FUNCTION_BLOCK Psd EXTENDS PlcModule
VAR_INPUT	
	Safety : Safety;
	
	{attribute 'OPC.UA.DA' := '0'}
	PsdConfig : PsdConfig;
	
	(* Axes *)
	IoStageAxis : IoStageAxis(Config := PsdConfig.AxesConfigs.IoStageAxisConfig);
	
	(* Chamber *)
	Chamber : PsdChamber(Config := PsdConfig.ChamberConfigs.PsdChamberConfig);
	
	(* Chuck *)
	Chuck : PsdChuck(Config := PsdConfig.ChuckConfigs.PsdChuckConfig);
	
	(* Ffu *)
	Ffu : Astrofan612Ffu(Config := PsdConfig.FfuConfigs.Astrofan612FfuConfig);
	
	(* Screen *)
	DM430GNScreenFS : DM430GNScreenFS(Config := PsdConfig.ScreenConfigs.DM430GNScreenConfigFS);
	DM430GNScreenBS : DM430GNScreenBS(Config := PsdConfig.ScreenConfigs.DM430GNScreenConfigBS);
	
	(* RFid *)
	Rfid : BisL405Rfid(Config := PsdConfig.RfidConfigs.BisL405RfidConfig);		
	
END_VAR
VAR_OUTPUT
END_VAR
VAR
END_VAR

SUPER^();

IF PsdConfig.SafetyIsEnabled THEN
	Safety();
END_IF

IF PsdConfig.AxesConfigs.IoStageAxisConfig.IsEnabled THEN
	IoStageAxis();	
END_IF

IF PsdConfig.ChamberConfigs.PsdChamberConfig.IsEnabled THEN
	Chamber();		
END_IF

IF PsdConfig.ChuckConfigs.PsdChuckConfig.IsEnabled THEN
	Chuck();		
END_IF

IF PsdConfig.FfuConfigs.Astrofan612FfuConfig.IsEnabled THEN
	Ffu();	
END_IF
	
// Screens
IF PsdConfig.ScreenConfigs.DM430GNScreenConfigFS.IsEnabled THEN
	DM430GNScreenFS();
	IF DM430GNScreenFS.InitConfigSerialCom THEN
		;
	END_IF
END_IF

IF PsdConfig.ScreenConfigs.DM430GNScreenConfigBS.IsEnabled THEN
	DM430GNScreenBS();
	IF DM430GNScreenBS.InitConfigSerialCom THEN
		;
	END_IF
END_IF

IF PsdConfig.RfidConfigs.BisL405RfidConfig.IsEnabled THEN
	Rfid();	
END_IF


IF IoStageAxis.GetPosition() = EStagePosition.Loading THEN
	Chamber.StageIsInLoadingPosition := TRUE;	
ELSE
	Chamber.StageIsInLoadingPosition := FALSE;
END_IF

METHOD FB_init : BOOL
VAR_INPUT
	bInitRetains : BOOL; // if TRUE, the retain variables are initialized (warm start / cold start)
	bInCopyCode : BOOL;  // if TRUE, the instance afterwards gets moved into the copy code (online change)
	Config : PsdConfig;
END_VAR
PsdConfig := Config;
PsdBkgrdSerialCom(Config := PsdConfig);

IF Config.IsEnabled THEN
	_logger.Information('Psd devices initialization starting...');
END_IF

// Axis
IF Config.AxesConfigs.IoStageAxisConfig.IsEnabled THEN
	IoStageAxis.FB_init(FALSE, FALSE, Config := Config.AxesConfigs.IoStageAxisConfig);	
END_IF

// Chamber
IF Config.ChamberConfigs.PsdChamberConfig.IsEnabled THEN
	Chamber.FB_init(FALSE, FALSE, Config := Config.ChamberConfigs.PsdChamberConfig);	
END_IF

// Chuck
IF Config.ChuckConfigs.PsdChuckConfig.IsEnabled THEN
	Chuck.FB_init(FALSE, FALSE, Config := Config.ChuckConfigs.PsdChuckConfig);	
END_IF

// FFU
IF Config.FfuConfigs.Astrofan612FfuConfig.IsEnabled THEN
	Ffu.FB_init(FALSE, FALSE, Config := Config.FfuConfigs.Astrofan612FfuConfig);	
END_IF

// Screens
IF Config.ScreenConfigs.DM430GNScreenConfigFS.IsEnabled THEN
	DM430GNScreenFS.FB_init(FALSE, FALSE, Config := Config.ScreenConfigs.DM430GNScreenConfigFS);	
END_IF
IF Config.ScreenConfigs.DM430GNScreenConfigBS.IsEnabled THEN
	DM430GNScreenBS.FB_init(FALSE, FALSE, Config := Config.ScreenConfigs.DM430GNScreenConfigBS);	
END_IF

// RFid
IF Config.RfidConfigs.BisL405RfidConfig.IsEnabled THEN
	Rfid.FB_init(FALSE, FALSE, Config := Config.RfidConfigs.BisL405RfidConfig);	
END_IF

IF Config.IsEnabled THEN
	_logger.Information('Psd devices initialization ended...');
END_IF
END_METHOD

END_FUNCTION_BLOCK

(* stored: Version 1.1.0.1, ProductVersion 3.1.4024.12
   POU Psd: Id {8356f6bd-4ce4-4674-aceb-72daafd0480c}, SpecialFunc None
   Method FB_init: Id {30401418-166a-40a2-a514-1027a884cb35} *)
